FUNCTION_BLOCK FB_A20
VAR_INPUT
END_VAR
VAR_OUTPUT
END_VAR
VAR
END_VAR

METHOD M_Stopping : M_Stopping
VAR_INPUT
END_VAR
END_METHOD

METHOD M_Test : BOOL
VAR_INPUT
END_VAR
//////////////add test here///////////////////////////
END_METHOD

END_FUNCTION_BLOCK

(* stored: Version 1.1.0.1, ProductVersion 3.1.4024.12
   POU FB_A20: Id {c114c468-3561-4b70-8115-825212b13cd3}, SpecialFunc None
   Method M_Stopping: Id {0ac067e4-610e-4b2e-b7a8-49c8a76ed805}
   Method M_Test: Id {1f305778-8145-43f9-93e1-f6337ff24382} *)
